{attribute addProperty BoxType "EJ2918-0000-0017"}
{attribute addProperty Id "FSoE_CommandUSINT811FSOUT_Module_1_Channel_1_OutputBIT10.1251FSOUT_Module_1_Channel_2_OutputBIT10.1252FSOUT_Module_1_Channel_3_OutputBIT10.1253FSOUT_Module_1_Channel_4_OutputBIT10.1254FSOUT_Module_1_ErrAckBIT10.1251FSOUT_Module_2_Channel_1_OutputBIT10.1251FSOUT_Module_2_Channel_2_OutputBIT10.1252FSOUT_Module_2_Channel_3_OutputBIT10.1253FSOUT_Module_2_Channel_4_OutputBIT10.1254FSOUT_Module_2_ErrAckBIT10.1251FSoE_CRC_000UINT1623FSoE_Connection_IDUINT1622"}
{attribute addProperty CRC "2310665834"}
{attribute addProperty SizeInBites "56"}
{attribute addProperty SizeInBytes "7"}
TYPE FSOE_89B9F66A :
STRUCT
	{attribute addProperty Name "FSoE_Command"}
	FSoE_Command : USINT;
	{attribute addProperty Name "FSOUT_Module_1_Channel_1_Output"}
	FSOUT_Module_1_Channel_1_Output : BIT;
	{attribute addProperty Name "FSOUT_Module_1_Channel_2_Output"}
	FSOUT_Module_1_Channel_2_Output : BIT;
	{attribute addProperty Name "FSOUT_Module_1_Channel_3_Output"}
	FSOUT_Module_1_Channel_3_Output : BIT;
	{attribute addProperty Name "FSOUT_Module_1_Channel_4_Output"}
	FSOUT_Module_1_Channel_4_Output : BIT;
	{attribute addProperty Name "FSOUT_Module_1_ErrAck"}
	FSOUT_Module_1_ErrAck : BIT;
	{attribute addProperty Name "FSOUT_Module_2_Channel_1_Output"}
	FSOUT_Module_2_Channel_1_Output : BIT;
	{attribute addProperty Name "FSOUT_Module_2_Channel_2_Output"}
	FSOUT_Module_2_Channel_2_Output : BIT;
	{attribute addProperty Name "FSOUT_Module_2_Channel_3_Output"}
	FSOUT_Module_2_Channel_3_Output : BIT;
	{attribute addProperty Name "FSOUT_Module_2_Channel_4_Output"}
	FSOUT_Module_2_Channel_4_Output : BIT;
	{attribute addProperty Name "FSOUT_Module_2_ErrAck"}
	FSOUT_Module_2_ErrAck : BIT;
	{attribute 'hide'}
	reserve_1_BIT_0 : BIT;
	{attribute 'hide'}
	reserve_1_BIT_1 : BIT;
	{attribute 'hide'}
	reserve_1_BIT_2 : BIT;
	{attribute 'hide'}
	reserve_1_BIT_3 : BIT;
	{attribute 'hide'}
	reserve_1_BIT_4 : BIT;
	{attribute 'hide'}
	reserve_1_BIT_5 : BIT;
	{attribute addProperty Name "FSoE_CRC_000"}
	FSoE_CRC_000 : UINT;
	{attribute addProperty Name "FSoE_Connection_ID"}
	FSoE_Connection_ID : UINT;
END_STRUCT
END_TYPE

(* stored: Version 1.2.0.0, ProductVersion 3.1.4024.9
   DUT FSOE_89B9F66A: Id {fc05ac3f-1967-483b-ac9f-d4d4a71a6fe6} *)
